TYPE ST_StaticSectorStatus :
STRUCT
	MoverIsOnSector			: BOOL;
	MoverCountOnSector		: UDINT;
	MoverEnteredSector		: Tc2_Standard.R_TRIG;
	MoverExitedSector		: Tc2_Standard.F_TRIG;
END_STRUCT
END_TYPE

(* stored: Version 1.1.0.1
   DUT ST_StaticSectorStatus: Id {81103d69-266a-0895-1575-10ee8e38fb8d} *)
